// TwinCAT 3 PLC project PLC1
// ProgramVersion: 3.1.4022.4
// libraries:
//   IO-Link Base, * (IO-Link)
//   SICK IOL WF_A70, * (SICK AG)
//   SICK IOL WLG4SC_3_A00, * (SICK AG)
//   Tc2_EtherCAT, * (Beckhoff Automation GmbH)
//   Tc2_Standard, * (Beckhoff Automation GmbH)
//   Tc2_System, * (Beckhoff Automation GmbH)
//   Tc3_Interfaces, * (Beckhoff Automation GmbH)
//   Tc3_Module, * (Beckhoff Automation GmbH)
// project tree:
//   / PlcTask.TcTTO
//   POUs/ MAIN.TcPOU
// real-time tasks:
//   TASK PlcTask: cycle T#10ms, priority 20, ADS port 350
// I/O:
//   DEVICE Device 2 (EtherCAT), AmsNetId 10.25.60.57.3.1
//     Box 1 (EPP1322-0001) [EPP1322-0001 3 port EtherCAT P gateway]
//     Box 2 (EPP6228-0022) [EPP6228 (IO Link Master)]
//       modules: Module 1 (DeviceState Inputs Device), Module 2 (DeviceState Inputs), Module 3 (IO-Link Slave), Module 4 (empty), Module 5 (empty), Module 6 (empty), Module 7 (empty), Module 8 (empty), Module 9 (empty), Module 10 (empty), Module 11 (Digital Inputs)
// variable links:
//   PLC1/PLC1 Instance <-> Device 2 (EtherCAT)
//     PlcTask Inputs/MAIN.startdata <-> Inputs/Frm0State

CONFIGURATION PLC1
    RESOURCE PLC ON TwinCAT3
        TASK PlcTask(INTERVAL := T#10ms, PRIORITY := 20);
        PROGRAM MAIN WITH PlcTask : MAIN;
    END_RESOURCE
END_CONFIGURATION

// ---- POUs/MAIN.TcPOU
PROGRAM MAIN
VAR		
	startdata 				AT %I* : UINT;	

	fbDemoAcyclic :			FB_SICK_WF_A70_EC;
	fbDemoProcesData :		FB_SICK_WF_A70_PB;
	structSick : 			ST_SICK_WF_A70;
	
	risingEdgeSignalRead : 		R_TRIG;
	risingEdgeSignalWrite :		R_TRIG;
	
	//Start read request
	xStartRead :			BOOL;
	
	//Start write request
	xStartWrite : 			BOOL;
	
	//Request done
	xDone :					BOOL;
	
END_VAR


risingEdgeSignalRead(CLK := xStartRead);
risingEdgeSignalWrite(CLK := xStartWrite);


structSick.Selection.AutoDeSelect := TRUE;

IF risingEdgeSignalRead.Q AND NOT fbDemoAcyclic.Busy THEN
	xDone := FALSE;
	structSick.Selection.ProductID := TRUE;
	structSick.Selection.VendorName := TRUE;
	structSick.Selection.ProductName := TRUE;
	structSick.Selection.KeyLock := TRUE;
	structSick.Selection.SwitchpointBDC1Q1.All := TRUE;
	
	fbDemoAcyclic.RW := FALSE; //Read
	fbDemoAcyclic.Req := TRUE; //Start job
	
	(*Parameter write*)
ELSIF risingEdgeSignalWrite.Q AND NOT fbDemoAcyclic.Busy THEN
	// Init status
	xDone:= FALSE;

	// Parameter selection that should be written
	structSick.Selection.KeyLock:= TRUE;
	
	
	// Definition of the data that should be written 
	structSick.Data.KeyLock:= eKeylock;

	
	fbDemoAcyclic.RW:= TRUE; // Write
	fbDemoAcyclic.Req:= TRUE; // Start job
END_IF;
	

fbDemoAcyclic(
	NetID:= '10.25.60.57.3.3', 
	PortNumber:= 1, 
	TimeOut:= T#5S, 
	Done=> , 
	Busy=> , 
	Error=> , 
	ErrorCode=> , 
	MasterType:= eBECKHOFF_6224, 
	SlaveAddr:= 0, 
	Req:= , 
	RW:= TRUE, 
	DeviceData:= structSick);
	
	fbDemoAcyclic.Req := FALSE;
	
	IF fbDemoAcyclic.Done THEN
		xDone := TRUE;
	END_IF

END_PROGRAM
